PROGRAM MAIN
VAR
    suite : FB_PidTests;
END_VAR

suite();
TcUnit.RUN();

END_PROGRAM

(* stored: Version 1.1.0.1
   POU MAIN: Id {72a389d0-e9a6-401b-a137-8089ca4cdeb1}, SpecialFunc None *)
